// TwinCAT 3 PLC project PLC
// ProgramVersion: 3.1.4024.0
// libraries:
//   EfficientIO Communicator, * (EfficientIO)
//   EfficientIO ModbusTCP, * (EfficientIO)
//   Lynus Energy Basic, * (Lynus AG)
//   Lynus Persistent Data V1, * (Lynus AG)
//   Tc2_ModbusSrv, * (Beckhoff Automation GmbH)
//   Tc2_Standard, * (Beckhoff Automation GmbH)
//   Tc2_System, * (Beckhoff Automation GmbH)
//   Tc2_Utilities, * (Beckhoff Automation GmbH)
//   Tc3_Module, * (Beckhoff Automation GmbH)
//   Lynus Standards,1.0.0.1,Lynus AG
// project tree:
//   / FastTask.TcTTO, MiddleTask.TcTTO, SlowTask.TcTTO
//   FB/ FB_Symo_PV_Inverter_FLOAT_1_DM_1_Inverter_1.TcPOU
//   POUs/ prgComEffIO.TcPOU, prgEM.TcPOU, prgPersistent.TcPOU, prgPV.TcPOU, prgRWEffIO.TcPOU, prgVarEffIO.TcPOU
// real-time tasks:
//   TASK FastTask: cycle T#5ms, priority 19, ADS port 351
//   TASK SlowTask: cycle T#20ms, priority 21, ADS port 352
//   TASK MiddleTask: cycle T#10ms, priority 20, ADS port 353
// I/O:
//   DEVICE Gerät 2 (CX-BK)
//     Box 1 (CX-BK)
// variable links:
//   PLC/PLC Instance <-> Device 2 (CX-BK)/Box 1 (CX-BK)
//     MiddleTask Inputs/prgEM.fbEM1.fbKL3403.byStateCH1 <-> Term 2 (KL3403)/Channel 1/Status
//     MiddleTask Inputs/prgEM.fbEM1.fbKL3403.byStateCH2 <-> Term 2 (KL3403)/Channel 2/Status
//     MiddleTask Inputs/prgEM.fbEM1.fbKL3403.byStateCH3 <-> Term 2 (KL3403)/Channel 3/Status
//     MiddleTask Inputs/prgEM.fbEM2.fbKL3403.byStateCH1 <-> Term 3 (KL3403)/Channel 1/Status
//     MiddleTask Inputs/prgEM.fbEM2.fbKL3403.byStateCH2 <-> Term 3 (KL3403)/Channel 2/Status
//     MiddleTask Inputs/prgEM.fbEM2.fbKL3403.byStateCH3 <-> Term 3 (KL3403)/Channel 3/Status
//     MiddleTask Inputs/prgEM.fbEM3.fbKL3403.byStateCH1 <-> Term 4 (KL3403)/Channel 1/Status
//     MiddleTask Inputs/prgEM.fbEM3.fbKL3403.byStateCH2 <-> Term 4 (KL3403)/Channel 2/Status
//     MiddleTask Inputs/prgEM.fbEM3.fbKL3403.byStateCH3 <-> Term 4 (KL3403)/Channel 3/Status
//     MiddleTask Inputs/prgEM.fbEM4.fbKL3403.byStateCH1 <-> Term 5 (KL3403)/Channel 1/Status
//     MiddleTask Inputs/prgEM.fbEM4.fbKL3403.byStateCH2 <-> Term 5 (KL3403)/Channel 2/Status
//     MiddleTask Inputs/prgEM.fbEM4.fbKL3403.byStateCH3 <-> Term 5 (KL3403)/Channel 3/Status
//     MiddleTask Inputs/prgEM.fbEM5.fbKL3403.byStateCH1 <-> Term 6 (KL3403)/Channel 1/Status
//     MiddleTask Inputs/prgEM.fbEM5.fbKL3403.byStateCH2 <-> Term 6 (KL3403)/Channel 2/Status
//     MiddleTask Inputs/prgEM.fbEM5.fbKL3403.byStateCH3 <-> Term 6 (KL3403)/Channel 3/Status
//     MiddleTask Inputs/prgEM.fbEM6.fbKL3403.byStateCH1 <-> Term 7 (KL3403)/Channel 1/Status
//     MiddleTask Inputs/prgEM.fbEM6.fbKL3403.byStateCH2 <-> Term 7 (KL3403)/Channel 2/Status
//     MiddleTask Inputs/prgEM.fbEM6.fbKL3403.byStateCH3 <-> Term 7 (KL3403)/Channel 3/Status
//     MiddleTask Inputs/prgEM.fbEM7.fbKL3403.byStateCH1 <-> Term 8 (KL3403)/Channel 1/Status
//     MiddleTask Inputs/prgEM.fbEM7.fbKL3403.byStateCH2 <-> Term 8 (KL3403)/Channel 2/Status
//     MiddleTask Inputs/prgEM.fbEM7.fbKL3403.byStateCH3 <-> Term 8 (KL3403)/Channel 3/Status
//     MiddleTask Inputs/prgEM.fbEM8.fbKL3403.byStateCH1 <-> Term 9 (KL3403)/Channel 1/Status
//     MiddleTask Inputs/prgEM.fbEM8.fbKL3403.byStateCH2 <-> Term 9 (KL3403)/Channel 2/Status
//     MiddleTask Inputs/prgEM.fbEM8.fbKL3403.byStateCH3 <-> Term 9 (KL3403)/Channel 3/Status
//     MiddleTask Inputs/prgEM.fbEM9.fbKL3403.byStateCH1 <-> Term 10 (KL3403)/Channel 1/Status
//     MiddleTask Inputs/prgEM.fbEM9.fbKL3403.byStateCH2 <-> Term 10 (KL3403)/Channel 2/Status
//     MiddleTask Inputs/prgEM.fbEM9.fbKL3403.byStateCH3 <-> Term 10 (KL3403)/Channel 3/Status
//     MiddleTask Inputs/prgEM.fbEM1.fbKL3403.iDataInCH1 <-> Term 2 (KL3403)/Channel 1/Daten Ein
//     MiddleTask Inputs/prgEM.fbEM1.fbKL3403.iDataInCH2 <-> Term 2 (KL3403)/Channel 2/Daten Ein
//     MiddleTask Inputs/prgEM.fbEM1.fbKL3403.iDataInCH3 <-> Term 2 (KL3403)/Channel 3/Daten Ein
//     MiddleTask Inputs/prgEM.fbEM2.fbKL3403.iDataInCH1 <-> Term 3 (KL3403)/Channel 1/Daten Ein
//     MiddleTask Inputs/prgEM.fbEM2.fbKL3403.iDataInCH2 <-> Term 3 (KL3403)/Channel 2/Daten Ein
//     MiddleTask Inputs/prgEM.fbEM2.fbKL3403.iDataInCH3 <-> Term 3 (KL3403)/Channel 3/Daten Ein
//     MiddleTask Inputs/prgEM.fbEM3.fbKL3403.iDataInCH1 <-> Term 4 (KL3403)/Channel 1/Daten Ein
//     MiddleTask Inputs/prgEM.fbEM3.fbKL3403.iDataInCH2 <-> Term 4 (KL3403)/Channel 2/Daten Ein
//     MiddleTask Inputs/prgEM.fbEM3.fbKL3403.iDataInCH3 <-> Term 4 (KL3403)/Channel 3/Daten Ein
//     MiddleTask Inputs/prgEM.fbEM4.fbKL3403.iDataInCH1 <-> Term 5 (KL3403)/Channel 1/Daten Ein
//     MiddleTask Inputs/prgEM.fbEM4.fbKL3403.iDataInCH2 <-> Term 5 (KL3403)/Channel 2/Daten Ein
//     MiddleTask Inputs/prgEM.fbEM4.fbKL3403.iDataInCH3 <-> Term 5 (KL3403)/Channel 3/Daten Ein
//     MiddleTask Inputs/prgEM.fbEM5.fbKL3403.iDataInCH1 <-> Term 6 (KL3403)/Channel 1/Daten Ein
//     MiddleTask Inputs/prgEM.fbEM5.fbKL3403.iDataInCH2 <-> Term 6 (KL3403)/Channel 2/Daten Ein
//     MiddleTask Inputs/prgEM.fbEM5.fbKL3403.iDataInCH3 <-> Term 6 (KL3403)/Channel 3/Daten Ein
//     MiddleTask Inputs/prgEM.fbEM6.fbKL3403.iDataInCH1 <-> Term 7 (KL3403)/Channel 1/Daten Ein
//     MiddleTask Inputs/prgEM.fbEM6.fbKL3403.iDataInCH2 <-> Term 7 (KL3403)/Channel 2/Daten Ein
//     MiddleTask Inputs/prgEM.fbEM6.fbKL3403.iDataInCH3 <-> Term 7 (KL3403)/Channel 3/Daten Ein
//     MiddleTask Inputs/prgEM.fbEM7.fbKL3403.iDataInCH1 <-> Term 8 (KL3403)/Channel 1/Daten Ein
//     MiddleTask Inputs/prgEM.fbEM7.fbKL3403.iDataInCH2 <-> Term 8 (KL3403)/Channel 2/Daten Ein
//     MiddleTask Inputs/prgEM.fbEM7.fbKL3403.iDataInCH3 <-> Term 8 (KL3403)/Channel 3/Daten Ein
//     MiddleTask Inputs/prgEM.fbEM8.fbKL3403.iDataInCH1 <-> Term 9 (KL3403)/Channel 1/Daten Ein
//     MiddleTask Inputs/prgEM.fbEM8.fbKL3403.iDataInCH2 <-> Term 9 (KL3403)/Channel 2/Daten Ein
//     MiddleTask Inputs/prgEM.fbEM8.fbKL3403.iDataInCH3 <-> Term 9 (KL3403)/Channel 3/Daten Ein
//     MiddleTask Inputs/prgEM.fbEM9.fbKL3403.iDataInCH1 <-> Term 10 (KL3403)/Channel 1/Daten Ein
//     MiddleTask Inputs/prgEM.fbEM9.fbKL3403.iDataInCH2 <-> Term 10 (KL3403)/Channel 2/Daten Ein
//     MiddleTask Inputs/prgEM.fbEM9.fbKL3403.iDataInCH3 <-> Term 10 (KL3403)/Channel 3/Daten Ein
//     MiddleTask Inputs/prgEM.fbKBusState.uiKBusState_OUT <-> Inputs/State
//     MiddleTask Outputs/prgEM.fbEM1.fbKL3403.byCntrCH1 <-> Term 2 (KL3403)/Channel 1/Kontrolle
//     MiddleTask Outputs/prgEM.fbEM1.fbKL3403.byCntrCH2 <-> Term 2 (KL3403)/Channel 2/Kontrolle
//     MiddleTask Outputs/prgEM.fbEM1.fbKL3403.byCntrCH3 <-> Term 2 (KL3403)/Channel 3/Kontrolle
//     MiddleTask Outputs/prgEM.fbEM2.fbKL3403.byCntrCH1 <-> Term 3 (KL3403)/Channel 1/Kontrolle
//     MiddleTask Outputs/prgEM.fbEM2.fbKL3403.byCntrCH2 <-> Term 3 (KL3403)/Channel 2/Kontrolle
//     MiddleTask Outputs/prgEM.fbEM2.fbKL3403.byCntrCH3 <-> Term 3 (KL3403)/Channel 3/Kontrolle
//     MiddleTask Outputs/prgEM.fbEM3.fbKL3403.byCntrCH1 <-> Term 4 (KL3403)/Channel 1/Kontrolle
//     MiddleTask Outputs/prgEM.fbEM3.fbKL3403.byCntrCH2 <-> Term 4 (KL3403)/Channel 2/Kontrolle
//     MiddleTask Outputs/prgEM.fbEM3.fbKL3403.byCntrCH3 <-> Term 4 (KL3403)/Channel 3/Kontrolle
//     MiddleTask Outputs/prgEM.fbEM4.fbKL3403.byCntrCH1 <-> Term 5 (KL3403)/Channel 1/Kontrolle
//     MiddleTask Outputs/prgEM.fbEM4.fbKL3403.byCntrCH2 <-> Term 5 (KL3403)/Channel 2/Kontrolle
//     MiddleTask Outputs/prgEM.fbEM4.fbKL3403.byCntrCH3 <-> Term 5 (KL3403)/Channel 3/Kontrolle
//     MiddleTask Outputs/prgEM.fbEM5.fbKL3403.byCntrCH1 <-> Term 6 (KL3403)/Channel 1/Kontrolle
//     MiddleTask Outputs/prgEM.fbEM5.fbKL3403.byCntrCH2 <-> Term 6 (KL3403)/Channel 2/Kontrolle
//     MiddleTask Outputs/prgEM.fbEM5.fbKL3403.byCntrCH3 <-> Term 6 (KL3403)/Channel 3/Kontrolle
//     MiddleTask Outputs/prgEM.fbEM6.fbKL3403.byCntrCH1 <-> Term 7 (KL3403)/Channel 1/Kontrolle
//     MiddleTask Outputs/prgEM.fbEM6.fbKL3403.byCntrCH2 <-> Term 7 (KL3403)/Channel 2/Kontrolle
//     MiddleTask Outputs/prgEM.fbEM6.fbKL3403.byCntrCH3 <-> Term 7 (KL3403)/Channel 3/Kontrolle
//     MiddleTask Outputs/prgEM.fbEM7.fbKL3403.byCntrCH1 <-> Term 8 (KL3403)/Channel 1/Kontrolle
//     MiddleTask Outputs/prgEM.fbEM7.fbKL3403.byCntrCH2 <-> Term 8 (KL3403)/Channel 2/Kontrolle
//     MiddleTask Outputs/prgEM.fbEM7.fbKL3403.byCntrCH3 <-> Term 8 (KL3403)/Channel 3/Kontrolle
//     MiddleTask Outputs/prgEM.fbEM8.fbKL3403.byCntrCH1 <-> Term 9 (KL3403)/Channel 1/Kontrolle
//     MiddleTask Outputs/prgEM.fbEM8.fbKL3403.byCntrCH2 <-> Term 9 (KL3403)/Channel 2/Kontrolle
//     MiddleTask Outputs/prgEM.fbEM8.fbKL3403.byCntrCH3 <-> Term 9 (KL3403)/Channel 3/Kontrolle
//     MiddleTask Outputs/prgEM.fbEM9.fbKL3403.byCntrCH1 <-> Term 10 (KL3403)/Channel 1/Kontrolle
//     MiddleTask Outputs/prgEM.fbEM9.fbKL3403.byCntrCH2 <-> Term 10 (KL3403)/Channel 2/Kontrolle
//     MiddleTask Outputs/prgEM.fbEM9.fbKL3403.byCntrCH3 <-> Term 10 (KL3403)/Channel 3/Kontrolle

CONFIGURATION PLC
    RESOURCE PLC ON TwinCAT3
        TASK FastTask(INTERVAL := T#5ms, PRIORITY := 19);
        TASK MiddleTask(INTERVAL := T#10ms, PRIORITY := 20);
        TASK SlowTask(INTERVAL := T#20ms, PRIORITY := 21);
        PROGRAM prgVarEffIO WITH FastTask : prgVarEffIO;
        PROGRAM prgRWEffIO WITH FastTask : prgRWEffIO;
        PROGRAM prgPersistent WITH FastTask : prgPersistent;
        PROGRAM prgEM WITH MiddleTask : prgEM;
        PROGRAM prgPV WITH MiddleTask : prgPV;
        PROGRAM prgComEffIO WITH SlowTask : prgComEffIO;
    END_RESOURCE
END_CONFIGURATION

// ---- POUs/prgVarEffIO.TcPOU
PROGRAM prgVarEffIO
VAR
	fbVar		: FB_VarInfo;
END_VAR

fbVar(
	bReadInfo:= , 
	eTMCFile:= eSelectTMCFile.eDontUseTMCFile, 
	eSavePositionTMCFile:= eSavePositionOnPLC.ePostionHardDisk, 
	udiCounterFoundVariables=> , 
	bError=> , 
	bBusy=> , 
	byProgress=> , 
	udiErrorCodeOut=> , 
	eErrorVarInfo_Out=> , 
	sVarWithError=> );
fbVar();
fbVar();

END_PROGRAM

// ---- POUs/prgRWEffIO.TcPOU
PROGRAM prgRWEffIO
VAR
	fbRW1		: FB_ReadWrite_V2;
	fbRW2		: FB_ReadWrite;
	fbRW3		: FB_ReadWrite;
	fbRW4		: FB_ReadWrite;
	i: INT;
	x: INT:=1;
END_VAR

fbRW1(	eUploadType := eSelectDataUploadType.e_Change_Intervall5min,
		bBusy=> , 
		bError=> , 
		udiErrorCodeOut=> , 
		eErrorReadWrite_Out=> );

fbRW2();
fbRW3();
fbRW4();

(*
FOR i:= 1 TO x BY 1 DO
	fbRW1();
	
END_FOR
*)

END_PROGRAM

// ---- POUs/prgPersistent.TcPOU
PROGRAM prgPersistent
VAR
	fbUSV		: FB_WritePersistentData_CX81xx;
	fb_Reboot		: NT_reboot;
	m_Reboot		: BOOL:=FALSE;
	ton_Auto_Reboot_Delay: Ton;
END_VAR

fbUSV(
	eSaveModeData:= eUSVSaveMode.eSaveWhenPowerfail, 
	bLoadPersistentDataOk=> , 
	bPowerFailDetect=> , 
	bError=> , 
	bySaveProcess=> , 
	dwStorageLast24h=> , 
	udiErrorCode=> );
	
		
fb_Reboot(	netid := '',
			delay := 2,
			start := m_Reboot OR ton_Auto_Reboot_Delay.Q);
			
ton_Auto_Reboot_Delay( 	In:= NOT prgComEffIO.fbCom.bConnected,
						PT := T#10M);

END_PROGRAM

// ---- POUs/prgComEffIO.TcPOU
PROGRAM prgComEffIO
VAR
	fbCom		: FB_MqttCommunicator_V2;
END_VAR

fbCom(
	bConnect:= TRUE, 
	strAuthkey := 'EIO08031879806',
	sUserName:= '0c3f05a0-7dc5-40a2-afb3-e4500c155bc7', 			
	sUserPassword:= '792aca21-1d48-4069-8bd7-51e04ad34ff6', 		
	eSavePositionCertificate:= eSavePositionOnPLC.ePostionHardDisk, 
	bConnected=> , 
	bError=> , 
	hrErrorCode=> , 
	eConnectionState=> , 
	eErrorMessage_Out=> );

END_PROGRAM

// ---- POUs/prgEM.TcPOU
PROGRAM prgEM
VAR
	fbKBusState		: FB_K_Bus_State;
	fbEM1			: FB_EM_Beckhoff_KL3403;
	fbEM1Counter	: FB_EnergyCounter;
	fbEM2			: FB_EM_Beckhoff_KL3403;
	fbEM2Counter	: FB_EnergyCounter;
	fbEM3			: FB_EM_Beckhoff_KL3403;
	fbEM3Counter	: FB_EnergyCounter;
	fbEM4			: FB_EM_Beckhoff_KL3403;
	fbEM4Counter	: FB_EnergyCounter;
	fbEM5			: FB_EM_Beckhoff_KL3403;
	fbEM5Counter	: FB_EnergyCounter;
	fbEM6			: FB_EM_Beckhoff_KL3403;
	fbEM6Counter	: FB_EnergyCounter;
	fbEM7			: FB_EM_Beckhoff_KL3403;
	fbEM7Counter	: FB_EnergyCounter;
	fbEM8			: FB_EM_Beckhoff_KL3403;
	fbEM8Counter	: FB_EnergyCounter;
	fbEM9			: FB_EM_Beckhoff_KL3403;
	fbEM9Counter	: FB_EnergyCounter;
	
	lrPowerEM1		: LREAL;						//{#lynus.ag#()}
	lrPowerEM2		: LREAL;						//{#lynus.ag#()}
	lrPowerEM3		: LREAL;						//{#lynus.ag#()}
	lrPowerEM4		: LREAL;						//{#lynus.ag#()}
	lrPowerEM5		: LREAL;						//{#lynus.ag#()}
	lrPowerEM6		: LREAL;						//{#lynus.ag#()}
	lrPowerEM7		: LREAL;						//{#lynus.ag#()}
	lrPowerEM8		: LREAL;						//{#lynus.ag#()}
	lrPowerEM9		: LREAL;						//{#lynus.ag#()}
	lrPowerEM9_Production	: LREAL;						//{#lynus.ag#()}
	lrPowerEM9_Consumption	: LREAL;						//{#lynus.ag#()}
	lr_InputVoltage_L1N		: LREAL;						//{#lynus.ag#()}
	lr_InputVoltage_L2N		: LREAL;						//{#lynus.ag#()}
	lr_InputVoltage_L3N		: LREAL;						//{#lynus.ag#()}
	lr_InputVoltage_L1L2	: LREAL;						//{#lynus.ag#()}
	lr_InputVoltage_L2L3	: LREAL;						//{#lynus.ag#()}
	lr_InputVoltage_L3L1	: LREAL;						//{#lynus.ag#()}
	lr_FrequencyEM1			: LREAL;						//{#lynus.ag#()}
	lr_CurrentL1EM1			: LREAL;						//{#lynus.ag#()}
	lr_CurrentL2EM1			: LREAL;						//{#lynus.ag#()}
	lr_CurrentL3EM1			: LREAL;						//{#lynus.ag#()}
	lrPower_RestAltbau		: LREAL;						//{#lynus.ag#()}
	lrPower_RestNeubau		: LREAL;						//{#lynus.ag#()}
	lrPower_FirmaGesamt		: LREAL;						//{#lynus.ag#()}
	fbRest_Altbau_Counter	: FB_EnergyCounter;
	fbRest_Neubau_Counter	: FB_EnergyCounter;
	fbFirmaGesamt_Counter	: FB_EnergyCounter;

END_VAR
VAR_INPUT
	uiCurrentTransformerRatio_EM1	:UINT:=300;			
	uiCurrentTransformerRatio_EM2	:UINT:=250;			
	uiCurrentTransformerRatio_EM3	:UINT:=250;
	uiCurrentTransformerRatio_EM4	:UINT:=200;
	uiCurrentTransformerRatio_EM5	:UINT:=100;
	uiCurrentTransformerRatio_EM6	:UINT:=150;
	uiCurrentTransformerRatio_EM7	:UINT:=1250;
	uiCurrentTransformerRatio_EM8	:UINT:=500;
	uiCurrentTransformerRatio_EM9	:UINT:=1000;
	mtest: BOOL;

END_VAR
VAR PERSISTENT
	lrCounterEM1	: LREAL;						//{#lynus.ag#()}
	lrCounterEM2	: LREAL;						//{#lynus.ag#()}
	lrCounterEM3	: LREAL;						//{#lynus.ag#()}
	lrCounterEM4	: LREAL;						//{#lynus.ag#()}
	lrCounterEM5	: LREAL;						//{#lynus.ag#()}
	lrCounterEM6	: LREAL;						//{#lynus.ag#()}
	lrCounterEM7	: LREAL;						//{#lynus.ag#()}
	lrCounterEM8	: LREAL;						//{#lynus.ag#()}
	lrCounterEM9	: LREAL;						//{#lynus.ag#()}
	lrCounter_Grid_Prod	: LREAL;						//{#lynus.ag#()}
	lrCounter_Grid_Cons	: LREAL;						//{#lynus.ag#()}
	lrCounterRestAltbau	: LREAL;						//{#lynus.ag#()}
	lrCounterRestNeubau	: LREAL;						//{#lynus.ag#()}
	lrCounterFirmaGesamt: LREAL;						//{#lynus.ag#()}
END_VAR

fbKBusState(	uiKBusState_OUT=> , 
				b_Kbus_notOk=> , 
				word_ErrorCount=> );


fbEM1(
	bEnable:= TRUE, 
	bChannel1Invers:= FALSE,
	bChannel2Invers:= FALSE,
	bChannel3Invers:= FALSE,
	uiCurrentTransformerRatioL1:= uiCurrentTransformerRatio_EM1, 
	uiCurrentTransformerRatioL2:= uiCurrentTransformerRatio_EM1, 
	uiCurrentTransformerRatioL3:= uiCurrentTransformerRatio_EM1, 
	uiKBusState_IN:= fbKBusState.uiKBusState_OUT, 
	stDataEMPower=> , 
	stDataEMCounter=> , 
	stDataEMPowerRealTime=> , 
	stDataEMCounterRealTime=> , 
	diNrOfEM_OUT=> );

lrPowerEM1 := fbEM1.stDataEMPower.lrPowerTotal;	
lr_InputVoltage_L1N := fbEM1.stDataEMPower.lrVoltageL1N;
lr_InputVoltage_L2N := fbEM1.stDataEMPower.lrVoltageL2N;
lr_InputVoltage_L3N := fbEM1.stDataEMPower.lrVoltageL3N;
lr_InputVoltage_L1L2 := fbEM1.stDataEMPower.lrVoltageL1L2;
lr_InputVoltage_L2L3 := fbEM1.stDataEMPower.lrVoltageL2L3;
lr_InputVoltage_L3L1 := fbEM1.stDataEMPower.lrVoltageL3L1;
lr_FrequencyEM1		:= fbEM1.stDataEMPower.lrFrequency;
lr_CurrentL1EM1		:= fbEM1.stDataEMPower.lrCurrentL1;
lr_CurrentL2EM1		:= fbEM1.stDataEMPower.lrCurrentL2;
lr_CurrentL3EM1		:= fbEM1.stDataEMPower.lrCurrentL3;

fbEM1Counter(
	byActiveTariff:= 1, 
	lrPowerInput:= lrPowerEM1, 
	lrTotalCounterEnergy_Consumption=> , 
	lrTotalCounterEnergy_Production=> , 
	lrCounterEnergyT1_Consumption=> , 
	lrCounterEnergyT2_Consumption=> , 
	lrCounterEnergyT1_Production=> , 
	lrCounterEnergyT2_Production=> );
	
IF fbEM1Counter.lrTotalCounterEnergy_Consumption > lrCounterEM1 THEN  	
	lrCounterEM1 := fbEM1Counter.lrTotalCounterEnergy_Consumption;
END_IF


fbEM2(
	bEnable:= TRUE, 
	bChannel1Invers:= FALSE,
	bChannel2Invers:= FALSE,
	bChannel3Invers:= FALSE,
	uiCurrentTransformerRatioL1:= uiCurrentTransformerRatio_EM2, 
	uiCurrentTransformerRatioL2:= uiCurrentTransformerRatio_EM2, 
	uiCurrentTransformerRatioL3:= uiCurrentTransformerRatio_EM2, 
	uiKBusState_IN:= fbKBusState.uiKBusState_OUT, 
	stDataEMPower=> , 
	stDataEMCounter=> , 
	stDataEMPowerRealTime=> , 
	stDataEMCounterRealTime=> , 
	diNrOfEM_OUT=> );

lrPowerEM2 := fbEM2.stDataEMPower.lrPowerTotal;	

fbEM2Counter(
	byActiveTariff:= 1, 
	lrPowerInput:= lrPowerEM2, 
	lrTotalCounterEnergy_Consumption=> , 
	lrTotalCounterEnergy_Production=> , 
	lrCounterEnergyT1_Consumption=> , 
	lrCounterEnergyT2_Consumption=> , 
	lrCounterEnergyT1_Production=> , 
	lrCounterEnergyT2_Production=> );
	
IF fbEM2Counter.lrTotalCounterEnergy_Consumption > lrCounterEM2 THEN  	
	lrCounterEM2 := fbEM2Counter.lrTotalCounterEnergy_Consumption;
END_IF


fbEM3(
	bEnable:= TRUE, 
	bChannel1Invers:= FALSE,
	bChannel2Invers:= FALSE,
	bChannel3Invers:= FALSE,
	uiCurrentTransformerRatioL1:= uiCurrentTransformerRatio_EM3, 
	uiCurrentTransformerRatioL2:= uiCurrentTransformerRatio_EM3, 
	uiCurrentTransformerRatioL3:= uiCurrentTransformerRatio_EM3, 
	uiKBusState_IN:= fbKBusState.uiKBusState_OUT, 
	stDataEMPower=> , 
	stDataEMCounter=> , 
	stDataEMPowerRealTime=> , 
	stDataEMCounterRealTime=> , 
	diNrOfEM_OUT=> );

lrPowerEM3 := fbEM3.stDataEMPower.lrPowerTotal;	

fbEM3Counter(
	byActiveTariff:= 1, 
	lrPowerInput:= lrPowerEM3, 
	lrTotalCounterEnergy_Consumption=> , 
	lrTotalCounterEnergy_Production=> , 
	lrCounterEnergyT1_Consumption=> , 
	lrCounterEnergyT2_Consumption=> , 
	lrCounterEnergyT1_Production=> , 
	lrCounterEnergyT2_Production=> );
	
IF fbEM3Counter.lrTotalCounterEnergy_Consumption > lrCounterEM3 THEN  	
	lrCounterEM3 := fbEM3Counter.lrTotalCounterEnergy_Consumption;
END_IF

fbEM4(
	bEnable:= TRUE, 
	bChannel1Invers:= FALSE,
	bChannel2Invers:= FALSE,
	bChannel3Invers:= FALSE,
	uiCurrentTransformerRatioL1:= uiCurrentTransformerRatio_EM4, 
	uiCurrentTransformerRatioL2:= uiCurrentTransformerRatio_EM4, 
	uiCurrentTransformerRatioL3:= uiCurrentTransformerRatio_EM4, 
	uiKBusState_IN:= fbKBusState.uiKBusState_OUT, 
	stDataEMPower=> , 
	stDataEMCounter=> , 
	stDataEMPowerRealTime=> , 
	stDataEMCounterRealTime=> , 
	diNrOfEM_OUT=> );

lrPowerEM4 := fbEM4.stDataEMPower.lrPowerTotal;	

fbEM4Counter(
	byActiveTariff:= 1, 
	lrPowerInput:= lrPowerEM4, 
	lrTotalCounterEnergy_Consumption=> , 
	lrTotalCounterEnergy_Production=> , 
	lrCounterEnergyT1_Consumption=> , 
	lrCounterEnergyT2_Consumption=> , 
	lrCounterEnergyT1_Production=> , 
	lrCounterEnergyT2_Production=> );
	
IF fbEM4Counter.lrTotalCounterEnergy_Consumption > lrCounterEM4 THEN  	
	lrCounterEM4 := fbEM4Counter.lrTotalCounterEnergy_Consumption;
END_IF

fbEM5(
	bEnable:= TRUE, 
	bChannel1Invers:= FALSE,
	bChannel2Invers:= FALSE,
	bChannel3Invers:= FALSE,
	uiCurrentTransformerRatioL1:= uiCurrentTransformerRatio_EM5, 
	uiCurrentTransformerRatioL2:= uiCurrentTransformerRatio_EM5, 
	uiCurrentTransformerRatioL3:= uiCurrentTransformerRatio_EM5, 
	uiKBusState_IN:= fbKBusState.uiKBusState_OUT, 
	stDataEMPower=> , 
	stDataEMCounter=> , 
	stDataEMPowerRealTime=> , 
	stDataEMCounterRealTime=> , 
	diNrOfEM_OUT=> );

lrPowerEM5 := fbEM5.stDataEMPower.lrPowerTotal;	

fbEM5Counter(
	byActiveTariff:= 1, 
	lrPowerInput:= lrPowerEM5, 
	lrTotalCounterEnergy_Consumption=> , 
	lrTotalCounterEnergy_Production=> , 
	lrCounterEnergyT1_Consumption=> , 
	lrCounterEnergyT2_Consumption=> , 
	lrCounterEnergyT1_Production=> , 
	lrCounterEnergyT2_Production=> );
	
IF fbEM5Counter.lrTotalCounterEnergy_Consumption > lrCounterEM5 THEN  	
	lrCounterEM5 := fbEM5Counter.lrTotalCounterEnergy_Consumption;
END_IF

fbEM6(
	bEnable:= TRUE, 
	bChannel1Invers:= FALSE,
	bChannel2Invers:= FALSE,
	bChannel3Invers:= FALSE,
	uiCurrentTransformerRatioL1:= uiCurrentTransformerRatio_EM6, 
	uiCurrentTransformerRatioL2:= uiCurrentTransformerRatio_EM6, 
	uiCurrentTransformerRatioL3:= uiCurrentTransformerRatio_EM6, 
	uiKBusState_IN:= fbKBusState.uiKBusState_OUT, 
	stDataEMPower=> , 
	stDataEMCounter=> , 
	stDataEMPowerRealTime=> , 
	stDataEMCounterRealTime=> , 
	diNrOfEM_OUT=> );

lrPowerEM6 := fbEM6.stDataEMPower.lrPowerTotal;	

fbEM6Counter(
	byActiveTariff:= 1, 
	lrPowerInput:= lrPowerEM6, 
	lrTotalCounterEnergy_Consumption=> , 
	lrTotalCounterEnergy_Production=> , 
	lrCounterEnergyT1_Consumption=> , 
	lrCounterEnergyT2_Consumption=> , 
	lrCounterEnergyT1_Production=> , 
	lrCounterEnergyT2_Production=> );
	
IF fbEM6Counter.lrTotalCounterEnergy_Consumption > lrCounterEM6 THEN  	
	lrCounterEM6 := fbEM6Counter.lrTotalCounterEnergy_Consumption;
END_IF

fbEM7(
	bEnable:= TRUE, 
	bChannel1Invers:= FALSE,
	bChannel2Invers:= FALSE,
	bChannel3Invers:= FALSE,
	uiCurrentTransformerRatioL1:= uiCurrentTransformerRatio_EM7, 
	uiCurrentTransformerRatioL2:= uiCurrentTransformerRatio_EM7, 
	uiCurrentTransformerRatioL3:= uiCurrentTransformerRatio_EM7, 
	uiKBusState_IN:= fbKBusState.uiKBusState_OUT, 
	stDataEMPower=> , 
	stDataEMCounter=> , 
	stDataEMPowerRealTime=> , 
	stDataEMCounterRealTime=> , 
	diNrOfEM_OUT=> );

lrPowerEM7 := fbEM7.stDataEMPower.lrPowerTotal;	

fbEM7Counter(
	byActiveTariff:= 1, 
	lrPowerInput:= lrPowerEM7, 
	lrTotalCounterEnergy_Consumption=> , 
	lrTotalCounterEnergy_Production=> , 
	lrCounterEnergyT1_Consumption=> , 
	lrCounterEnergyT2_Consumption=> , 
	lrCounterEnergyT1_Production=> , 
	lrCounterEnergyT2_Production=> );
	
IF fbEM7Counter.lrTotalCounterEnergy_Consumption > lrCounterEM7 THEN  	
	lrCounterEM7 := fbEM7Counter.lrTotalCounterEnergy_Consumption;
END_IF

fbEM8(
	bEnable:= TRUE, 
	bChannel1Invers:= FALSE,
	bChannel2Invers:= FALSE,
	bChannel3Invers:= FALSE,
	uiCurrentTransformerRatioL1:= uiCurrentTransformerRatio_EM8, 
	uiCurrentTransformerRatioL2:= uiCurrentTransformerRatio_EM8, 
	uiCurrentTransformerRatioL3:= uiCurrentTransformerRatio_EM8, 
	uiKBusState_IN:= fbKBusState.uiKBusState_OUT, 
	stDataEMPower=> , 
	stDataEMCounter=> , 
	stDataEMPowerRealTime=> , 
	stDataEMCounterRealTime=> , 
	diNrOfEM_OUT=> );

lrPowerEM8 := fbEM8.stDataEMPower.lrPowerTotal;	

fbEM8Counter(
	byActiveTariff:= 1, 
	lrPowerInput:= lrPowerEM8, 
	lrTotalCounterEnergy_Consumption=> , 
	lrTotalCounterEnergy_Production=> , 
	lrCounterEnergyT1_Consumption=> , 
	lrCounterEnergyT2_Consumption=> , 
	lrCounterEnergyT1_Production=> , 
	lrCounterEnergyT2_Production=> );
	
IF fbEM8Counter.lrTotalCounterEnergy_Consumption > lrCounterEM8 THEN  	
	lrCounterEM8 := fbEM8Counter.lrTotalCounterEnergy_Consumption;
END_IF

fbEM9(
	bEnable:= TRUE, 
	bChannel1Invers:= FALSE,
	bChannel2Invers:= FALSE,
	bChannel3Invers:= FALSE,
	uiCurrentTransformerRatioL1:= uiCurrentTransformerRatio_EM9, 
	uiCurrentTransformerRatioL2:= uiCurrentTransformerRatio_EM9, 
	uiCurrentTransformerRatioL3:= uiCurrentTransformerRatio_EM9, 
	uiKBusState_IN:= fbKBusState.uiKBusState_OUT, 
	stDataEMPower=> , 
	stDataEMCounter=> , 
	stDataEMPowerRealTime=> , 
	stDataEMCounterRealTime=> , 
	diNrOfEM_OUT=> );

lrPowerEM9 := fbEM9.stDataEMPower.lrPowerTotal;	

IF lrPowerEM9<= 0 THEN
	lrPowerEM9_Production :=  lrPowerEM9;
	lrPowerEM9_Consumption := 0;
ELSE
	lrPowerEM9_Production :=  0;
	lrPowerEM9_Consumption := lrPowerEM9;
END_IF

fbEM9Counter(
	byActiveTariff:= 1, 
	lrPowerInput:= lrPowerEM9, 
	lrTotalCounterEnergy_Consumption=> , 
	lrTotalCounterEnergy_Production=> , 
	lrCounterEnergyT1_Consumption=> , 
	lrCounterEnergyT2_Consumption=> , 
	lrCounterEnergyT1_Production=> , 
	lrCounterEnergyT2_Production=> );
	
IF fbEM9Counter.lrTotalCounterEnergy_Consumption > lrCounterEM9 THEN  	
	lrCounterEM9 := fbEM9Counter.lrTotalCounterEnergy_Consumption;
	lrCounter_Grid_Cons	:= fbEM9Counter.lrTotalCounterEnergy_Consumption;
END_IF

IF fbEM9Counter.lrTotalCounterEnergy_Production > lrCounter_Grid_Prod THEN  	
	lrCounter_Grid_Prod := fbEM9Counter.lrTotalCounterEnergy_Production;
END_IF

lrPower_RestAltbau := lrPowerEM8 - lrPowerEM1 - lrPowerEM2 - lrPowerEM3 - lrPowerEM4 + prgPV.lrPowerPV;
lrPower_RestAltbau := LIMIT(0,lrPower_RestAltbau,lrPower_RestAltbau);
lrPower_RestNeubau := lrPowerEM9 - lrPowerEM8 - lrPowerEM5 - lrPowerEM6;
lrPower_RestNeubau := LIMIT(0,lrPower_RestNeubau,lrPower_RestNeubau);

lrPower_FirmaGesamt := lrPowerEM9 + prgPV.lrPowerPV;


fbRest_Altbau_Counter(
	byActiveTariff:= 1, 
	lrPowerInput:= lrPower_RestAltbau, 
	lrTotalCounterEnergy_Consumption=> , 
	lrTotalCounterEnergy_Production=> , 
	lrCounterEnergyT1_Consumption=> , 
	lrCounterEnergyT2_Consumption=> , 
	lrCounterEnergyT1_Production=> , 
	lrCounterEnergyT2_Production=> );
	
IF fbRest_Altbau_Counter.lrTotalCounterEnergy_Consumption > lrCounterRestAltbau THEN  	
	lrCounterRestAltbau := fbRest_Altbau_Counter.lrTotalCounterEnergy_Consumption;
END_IF


fbRest_Neubau_Counter(
	byActiveTariff:= 1, 
	lrPowerInput:= lrPower_RestNeubau, 
	lrTotalCounterEnergy_Consumption=> , 
	lrTotalCounterEnergy_Production=> , 
	lrCounterEnergyT1_Consumption=> , 
	lrCounterEnergyT2_Consumption=> , 
	lrCounterEnergyT1_Production=> , 
	lrCounterEnergyT2_Production=> );
	
IF fbRest_Neubau_Counter.lrTotalCounterEnergy_Consumption > lrCounterRestNeubau THEN  	
	lrCounterRestNeubau := fbRest_Neubau_Counter.lrTotalCounterEnergy_Consumption;
END_IF


fbFirmaGesamt_Counter(
	byActiveTariff:= 1, 
	lrPowerInput:= lrPower_FirmaGesamt, 
	lrTotalCounterEnergy_Consumption=> , 
	lrTotalCounterEnergy_Production=> , 
	lrCounterEnergyT1_Consumption=> , 
	lrCounterEnergyT2_Consumption=> , 
	lrCounterEnergyT1_Production=> , 
	lrCounterEnergyT2_Production=> );
	
IF fbFirmaGesamt_Counter.lrTotalCounterEnergy_Consumption > lrCounterFirmaGesamt THEN  	
	lrCounterFirmaGesamt := fbFirmaGesamt_Counter.lrTotalCounterEnergy_Consumption;
END_IF

END_PROGRAM

// ---- POUs/prgPV.TcPOU
PROGRAM prgPV
VAR
	fbPV_1					: FB_Symo_PV_Inverter_float_1_DM_1_Inverter_1;
	fbPV_2					: FB_Symo_PV_Inverter_float_1_DM_1_Inverter_1;
	fbPV_3					: FB_Symo_PV_Inverter_float_1_DM_1_Inverter_1;
	fbPV_4					: FB_Symo_PV_Inverter_float_1_DM_1_Inverter_1;
	fbPV_5					: FB_Symo_PV_Inverter_float_1_DM_1_Inverter_1;
	fbPV_6					: FB_Symo_PV_Inverter_float_1_DM_1_Inverter_1;
	fbPV_7					: FB_Symo_PV_Inverter_float_1_DM_1_Inverter_1;
	fbPV_8					: FB_Symo_PV_Inverter_float_1_DM_1_Inverter_1;
	lrPowerPV				: LREAL;				//{#lynus.ag#()}
	lrPowerPV_1				: LREAL;				//{#lynus.ag#()}
	lrPowerPV_2				: LREAL;				//{#lynus.ag#()}
	lrPowerPV_3				: LREAL;				//{#lynus.ag#()}
	lrPowerPV_4				: LREAL;				//{#lynus.ag#()}
	lrPowerPV_5				: LREAL;				//{#lynus.ag#()}
	lrPowerPV_6				: LREAL;				//{#lynus.ag#()}
	lrPowerPV_7				: LREAL;				//{#lynus.ag#()}
	lrPowerPV_8				: LREAL;				//{#lynus.ag#()}
	fbCounterPV_1			: FB_EnergyCounter;
	fbCounterPV_2			: FB_EnergyCounter;
	fbCounterPV_3			: FB_EnergyCounter;
	fbCounterPV_4			: FB_EnergyCounter;
	fbCounterPV_5			: FB_EnergyCounter;
	fbCounterPV_6			: FB_EnergyCounter;
	fbCounterPV_7			: FB_EnergyCounter;
	fbCounterPV_8			: FB_EnergyCounter;
	fbCounterPV				: FB_EnergyCounter;
END_VAR
VAR PERSISTENT
	lrCounterPV_1	: LREAL;						//{#lynus.ag#()}
	lrCounterPV_2	: LREAL;						//{#lynus.ag#()}
	lrCounterPV_3	: LREAL;						//{#lynus.ag#()}
	lrCounterPV_4	: LREAL;						//{#lynus.ag#()}
	lrCounterPV_5	: LREAL;						//{#lynus.ag#()}
	lrCounterPV_6	: LREAL;						//{#lynus.ag#()}
	lrCounterPV_7	: LREAL;						//{#lynus.ag#()}
	lrCounterPV_8	: LREAL;						//{#lynus.ag#()}
	lrCounterPV		: LREAL;						//{#lynus.ag#()}
	m_Enable_PV1: BOOL:= TRUE;
	m_Enable_PV2: BOOL:= true;
	m_Enable_PV3: BOOL:= true;
	m_Enable_PV4: BOOL:= true;
	m_Enable_PV5: BOOL:= true;
	m_Enable_PV6: BOOL:= true;
	m_Enable_PV7: BOOL:= true;
	m_Enable_PV8: BOOL:= true;	

END_VAR

fbPV_1(
	bEnable:= TRUE, 
	sIPAdress:= '192.168.10.12', 
	byUnitID_Inverter:=3 , 
	stDataSymo10=> , 
	stDataEMPower_PV=> , 
	stDataEMCounter_PV=> , 
	diNrOfEM_OUT_PV=> );
lrPowerPV_1 := fbPV_1.stDataEMPower_PV.lrPowerTotal;
fbPV_2(
	bEnable:= m_Enable_PV2, 
	sIPAdress:= '192.168.10.13', 
	byUnitID_Inverter:=2 , 
	stDataSymo10=> , 
	stDataEMPower_PV=> , 
	stDataEMCounter_PV=> , 
	diNrOfEM_OUT_PV=> );
lrPowerPV_2 := fbPV_2.stDataEMPower_PV.lrPowerTotal;
fbPV_3(
	bEnable:= m_Enable_PV3, 
	sIPAdress:= '192.168.10.14', 
	byUnitID_Inverter:=5 , 
	stDataSymo10=> , 
	stDataEMPower_PV=> , 
	stDataEMCounter_PV=> , 
	diNrOfEM_OUT_PV=> );
lrPowerPV_3 := fbPV_3.stDataEMPower_PV.lrPowerTotal;
fbPV_4(
	bEnable:= m_Enable_PV4, 
	sIPAdress:= '192.168.10.15', 
	byUnitID_Inverter:=4 , 
	stDataSymo10=> , 
	stDataEMPower_PV=> , 
	stDataEMCounter_PV=> , 
	diNrOfEM_OUT_PV=> );
lrPowerPV_4 := fbPV_4.stDataEMPower_PV.lrPowerTotal;
fbPV_5(
	bEnable:= m_Enable_PV5, 
	sIPAdress:= '192.168.10.16', 
	byUnitID_Inverter:=1 , 
	stDataSymo10=> , 
	stDataEMPower_PV=> , 
	stDataEMCounter_PV=> , 
	diNrOfEM_OUT_PV=> );
lrPowerPV_5 := fbPV_5.stDataEMPower_PV.lrPowerTotal;
fbPV_6(
	bEnable:= m_Enable_PV6, 
	sIPAdress:= '192.168.10.17', 
	byUnitID_Inverter:=1 , 
	stDataSymo10=> , 
	stDataEMPower_PV=> , 
	stDataEMCounter_PV=> , 
	diNrOfEM_OUT_PV=> );
lrPowerPV_6 := fbPV_6.stDataEMPower_PV.lrPowerTotal;
fbPV_7(
	bEnable:= m_Enable_PV7, 
	sIPAdress:= '192.168.10.18', 
	byUnitID_Inverter:=1 , 
	stDataSymo10=> , 
	stDataEMPower_PV=> , 
	stDataEMCounter_PV=> , 
	diNrOfEM_OUT_PV=> );
lrPowerPV_7 := fbPV_7.stDataEMPower_PV.lrPowerTotal;
fbPV_8(
	bEnable:= m_Enable_PV8, 
	sIPAdress:= '192.168.10.19', 
	byUnitID_Inverter:=1 , 
	stDataSymo10=> , 
	stDataEMPower_PV=> , 
	stDataEMCounter_PV=> , 
	diNrOfEM_OUT_PV=> );
lrPowerPV_8 := fbPV_8.stDataEMPower_PV.lrPowerTotal;

lrPowerPV := lrPowerPV_1 + lrPowerPV_2 + lrPowerPV_3 + lrPowerPV_4 + lrPowerPV_5 + lrPowerPV_6 + lrPowerPV_7 + lrPowerPV_8;


// kWh Counters

fbCounterPV_1(
	byActiveTariff:= 1, 
	lrPowerInput:= lrPowerPV_1, 
	lrTotalCounterEnergy_Consumption=> , 
	lrTotalCounterEnergy_Production=> , 
	lrCounterEnergyT1_Consumption=> , 
	lrCounterEnergyT2_Consumption=> , 
	lrCounterEnergyT1_Production=> , 
	lrCounterEnergyT2_Production=> );
	
IF fbCounterPV_1.lrTotalCounterEnergy_Consumption > lrCounterPV_1 THEN  	
	lrCounterPV_1 := fbCounterPV_1.lrTotalCounterEnergy_Consumption;
END_IF

fbCounterPV_2(
	byActiveTariff:= 1, 
	lrPowerInput:= lrPowerPV_2, 
	lrTotalCounterEnergy_Consumption=> , 
	lrTotalCounterEnergy_Production=> , 
	lrCounterEnergyT1_Consumption=> , 
	lrCounterEnergyT2_Consumption=> , 
	lrCounterEnergyT1_Production=> , 
	lrCounterEnergyT2_Production=> );
	
IF fbCounterPV_2.lrTotalCounterEnergy_Consumption > lrCounterPV_2 THEN  	
	lrCounterPV_2 := fbCounterPV_2.lrTotalCounterEnergy_Consumption;
END_IF

fbCounterPV_3(
	byActiveTariff:= 1, 
	lrPowerInput:= lrPowerPV_3, 
	lrTotalCounterEnergy_Consumption=> , 
	lrTotalCounterEnergy_Production=> , 
	lrCounterEnergyT1_Consumption=> , 
	lrCounterEnergyT2_Consumption=> , 
	lrCounterEnergyT1_Production=> , 
	lrCounterEnergyT2_Production=> );
	
IF fbCounterPV_3.lrTotalCounterEnergy_Consumption > lrCounterPV_3 THEN  	
	lrCounterPV_3 := fbCounterPV_3.lrTotalCounterEnergy_Consumption;
END_IF

fbCounterPV_4(
	byActiveTariff:= 1, 
	lrPowerInput:= lrPowerPV_4, 
	lrTotalCounterEnergy_Consumption=> , 
	lrTotalCounterEnergy_Production=> , 
	lrCounterEnergyT1_Consumption=> , 
	lrCounterEnergyT2_Consumption=> , 
	lrCounterEnergyT1_Production=> , 
	lrCounterEnergyT2_Production=> );
	
IF fbCounterPV_4.lrTotalCounterEnergy_Consumption > lrCounterPV_4 THEN  	
	lrCounterPV_4 := fbCounterPV_4.lrTotalCounterEnergy_Consumption;
END_IF

fbCounterPV_5(
	byActiveTariff:= 1, 
	lrPowerInput:= lrPowerPV_5, 
	lrTotalCounterEnergy_Consumption=> , 
	lrTotalCounterEnergy_Production=> , 
	lrCounterEnergyT1_Consumption=> , 
	lrCounterEnergyT2_Consumption=> , 
	lrCounterEnergyT1_Production=> , 
	lrCounterEnergyT2_Production=> );
	
IF fbCounterPV_5.lrTotalCounterEnergy_Consumption > lrCounterPV_5 THEN  	
	lrCounterPV_5 := fbCounterPV_5.lrTotalCounterEnergy_Consumption;
END_IF

fbCounterPV_6(
	byActiveTariff:= 1, 
	lrPowerInput:= lrPowerPV_6, 
	lrTotalCounterEnergy_Consumption=> , 
	lrTotalCounterEnergy_Production=> , 
	lrCounterEnergyT1_Consumption=> , 
	lrCounterEnergyT2_Consumption=> , 
	lrCounterEnergyT1_Production=> , 
	lrCounterEnergyT2_Production=> );
	
IF fbCounterPV_6.lrTotalCounterEnergy_Consumption > lrCounterPV_6 THEN  	
	lrCounterPV_6 := fbCounterPV_6.lrTotalCounterEnergy_Consumption;
END_IF

fbCounterPV_7(
	byActiveTariff:= 1, 
	lrPowerInput:= lrPowerPV_7, 
	lrTotalCounterEnergy_Consumption=> , 
	lrTotalCounterEnergy_Production=> , 
	lrCounterEnergyT1_Consumption=> , 
	lrCounterEnergyT2_Consumption=> , 
	lrCounterEnergyT1_Production=> , 
	lrCounterEnergyT2_Production=> );
	
IF fbCounterPV_7.lrTotalCounterEnergy_Consumption > lrCounterPV_7 THEN  	
	lrCounterPV_7 := fbCounterPV_7.lrTotalCounterEnergy_Consumption;
END_IF

fbCounterPV_8(
	byActiveTariff:= 1, 
	lrPowerInput:= lrPowerPV_8, 
	lrTotalCounterEnergy_Consumption=> , 
	lrTotalCounterEnergy_Production=> , 
	lrCounterEnergyT1_Consumption=> , 
	lrCounterEnergyT2_Consumption=> , 
	lrCounterEnergyT1_Production=> , 
	lrCounterEnergyT2_Production=> );
	
IF fbCounterPV_8.lrTotalCounterEnergy_Consumption > lrCounterPV_8 THEN  	
	lrCounterPV_8 := fbCounterPV_8.lrTotalCounterEnergy_Consumption;
END_IF

fbCounterPV(
	byActiveTariff:= 1, 
	lrPowerInput:= lrPowerPV, 
	lrTotalCounterEnergy_Consumption=> , 
	lrTotalCounterEnergy_Production=> , 
	lrCounterEnergyT1_Consumption=> , 
	lrCounterEnergyT2_Consumption=> , 
	lrCounterEnergyT1_Production=> , 
	lrCounterEnergyT2_Production=> );
	
IF fbCounterPV.lrTotalCounterEnergy_Consumption > lrCounterPV THEN  	
	lrCounterPV := fbCounterPV.lrTotalCounterEnergy_Consumption;
END_IF

END_PROGRAM

// ---- FB/FB_Symo_PV_Inverter_FLOAT_1_DM_1_Inverter_1.TcPOU
{attribute 'hide_all_locals'}
FUNCTION_BLOCK FB_Symo_PV_Inverter_FLOAT_1_DM_1_Inverter_1
VAR_INPUT PERSISTENT
	bEnable						: BOOL;												//True = Function is enabled, FALSE = Function is dissabled, no new Data
	sIPAdress					: STRING(15);										//IP Adress from the Inverter
	byUnitID_Inverter			: BYTE;												//Unit ID fromt the Inverter (1 to 247)
END_VAR
VAR_OUTPUT
	stDataSymo10				: ST_Symo_PV_OutData;								//Output structure with Data from Symo 10
	stDataEMPower_PV			: ST_ElectricMeter_Output_Power;					//Output structure with Data from Electric Meter PV (Power Data)
	stDataEMCounter_PV			: ST_ElectricMeter_Output_Counter;					//Output structure with Data from Electric Meter PV (Counter Data)
	diNrOfEM_OUT_PV				: DINT;												//Active Number from the Electric Meter for using on other functions
END_VAR
VAR
	fbElMeter					: FB_ElectricMeter;									//Electric Meter Function 
	fbNumberDevice				: FB_NumberOfDevice;								//Function block to calcualte the number of the Device
	fbConvertEnergyRegister		: FB_CV_WORD_TO_DWORD;								//Convert function
	fbMBRead_FC3				: FB_MBReadRegs;									//Modbus Read Function (FC3)
	timDelay					: TON;												//Timer for Delay between Requests
	timTimeout					: TON;												//Timer for Timeout
	timDissableFunctions		: TON;												//Timer to dissable the Function after Lynus_Standards.Constants_General.tTimeDissableLynusFunctions Days without connection to the Lynus Cloud
	timResetConnectionOnGVL		: TON;												//Timer to try reset the connection Flag on the GVL. (When somebody delete the Connection Function and make only a onlinechange)
	FPEnable					: R_TRIG;											//Internal positive Edge
	FPError_FC_3				: R_TRIG;											//Internal positive Edge
	PD_String					: FB_PersistentData_String;							//Function to save persistent data 
	stFloat						: ST_UN_FLOAT_CONVERT_DWORD_REAL;					//Convert the Float Raw Value
	arrBuffer_FC3				: ARRAY[1..47] OF WORD;								//Buffer with Data from FC3
	arrPD						: ARRAY[1..2] OF FB_PersistentData_Number;			//Function to save persistent data 
	byWaitInStep				: BYTE;												//Wait in Step before start to clean data on PLC
	iStateGVLData				: INT;												//State machine to handle the data on the GVL
	iStateModbus				: INT;												//State variable for Statemachine
	iStateModbus_CP				: INT;												//Compare State variable
	diCounterForGVL				: DINT;												//Counter to clean old data on GVL
	lrCheckValue				: LREAL;											//Internal Value to check the value before convert
END_VAR

//Creator : Kai Ebensperger
//Company : Lynus AG
//Date : 28.04.2021
//Version : 1.0.0.0

//With this function its possible to read out values from the Symo 10 PV Inverter from the factory Fronius
//This Function read out the Values from 1 Fronius Datamanager with maximal 1 Inverter.
//The protocol to the Inverter is Modbus TCP
//Versions that are supported : 1.1.5-0
//Attention. To access the registers, an offset of 1 must always be subtracted. Register 40001 would then be on register 40000.
//This Function use the FLOAT Format

//NOTE for diNr.....Designation => 
//_IN = Here Data come in from other Functions or go out to other functions about the GVL
//_OUT = Here Data go out to other functions about the GVL

(*------------------------------------------------------------------------------------------General Input Part---------------------------------------------------------------------------------------------*)

//Check limitation
byUnitID_Inverter := LIMIT(1,byUnitID_Inverter,247);

(*-------------------------------------------------------------Calcualte the number of EM System---------------------------------------------------------------*)

fbNumberDevice(
	diActualNumberOfDevices:= Lynus_Standards.GVL_Energy.stNumberOfDevices.diNumberOfElectricMeters, 
	diMaxNumberOfDevices:= Constants_Energy.diMaxNumberOfElectricMeters, 
	udiCounterOnlineChange:= TwinCAT_SystemInfoVarList._AppInfo.OnlineChangeCnt, 
	bNumberIsCalculatet=> , 
	bFPNumberIsCalculatet=> , 
	bOnlineChange=> , 
	diNumberForThisDevice=> diNrOfEM_OUT_PV, 
	diNumberOfTotalDevices=> );

//Write new Numer on GVL
IF fbNumberDevice.bFPNumberIsCalculatet THEN
	Lynus_Standards.GVL_Energy.stNumberOfDevices.diNumberOfElectricMeters := fbNumberDevice.diNumberOfTotalDevices;	
END_IF 

//Delete old Number on GVL
IF fbNumberDevice.bOnlineChange THEN 
	Lynus_Standards.GVL_Energy.stNumberOfDevices.diNumberOfElectricMeters := diNrOfEM_OUT_PV;	
		iStateGVLData := 1; 
END_IF

(*-------------------------------------------------------------Service from Backend is ready and check the connection to backen for dissabel/enable Function---------------------------------------------------------------*)

//Try to reset the variable for connection on the GVL. When all is normal then the Lynus Mqtt connection function set this variable to true in the next cycle
//When we have no connection to the backend then after Lynus_Standards.Constants_General.tTimeDissableLynusFunctions days the Function is dissabled with all of his functionalities
timResetConnectionOnGVL(IN:= NOT timResetConnectionOnGVL.Q, PT:= T#1H, Q=> , ET=> );
	IF timResetConnectionOnGVL.Q THEN Lynus_Standards.GVL_Communicator.bStateConnectionToEnableFunctions := FALSE; END_IF
		IF NOT Lynus_Standards.GVL_Communicator.bStateConnectionToEnableFunctions THEN timDissableFunctions.IN := TRUE; ELSE timDissableFunctions.IN := FALSE; END_IF  
			timDissableFunctions(IN:= , PT:= Lynus_Standards.Constants_General.tTimeDissableLynusFunctions, Q=> , ET=> );
	
(*------------------------------------------------------------------------------------------State Machine---------------------------------------------------------------------------------------------*)
	
//Enable
FPEnable(CLK:= bEnable, Q=> );
	IF FPEnable.Q AND iStateModbus = 0 THEN iStateModbus := 1; END_IF
		IF NOT bEnable OR timDissableFunctions.Q THEN iStateModbus := 0; END_IF

//Timer for delay
timDelay(IN:= , PT:= T#100MS, Q=> , ET=> );	

//Timer for Timeout in Statemachine
	IF iStateModbus = iStateModbus_CP THEN timTimeout.IN := TRUE; ELSE timTimeout.IN := FALSE; END_IF
		IF iStateModbus = 0 THEN timTimeout.IN := FALSE; END_IF
timTimeout(IN:= , PT:= T#20S, Q=> , ET=> );	

//Statemachine
CASE iStateModbus OF
	
	0://Init Step
		iStateModbus_CP := iStateModbus;
			timDelay.IN := FALSE;
		
		stDataSymo10.bFunctionIsActive := FALSE;
			stDataSymo10.eOperatingStateInverter := E_Symo_PV_OperatingState.eNoDataReceived;
				fbMBRead_FC3.bExecute := FALSE;
					lrCheckValue := 0;
									
	1://Read out first Registers from 40072 to 40118
		stDataSymo10.bFunctionIsActive := TRUE;
			iStateModbus_CP := iStateModbus;
		
		fbMBRead_FC3.nQuantity := 47;
			fbMBRead_FC3.nMBAddr := 40071;
				fbMBRead_FC3.bExecute := TRUE;
					fbMBRead_FC3.nUnitID := byUnitID_Inverter;
			
		IF fbMBRead_FC3.bBusy THEN timDelay.IN := TRUE; END_IF
		
		//Wait for Delay, copy Data and then next step
		IF NOT fbMBRead_FC3.bBusy AND NOT fbMBRead_FC3.bError AND timDelay.Q THEN
			//Copy Data Current L1
			fbConvertEnergyRegister(wInputValue_1:= arrBuffer_FC3[3], wInputValue_2:= arrBuffer_FC3[4], eByteOrderForConvert:= eByteOrder.eBigEndian, dwOutputValue=> );
				stFloat.dwRawValue := fbConvertEnergyRegister.dwOutputValue;
					lrCheckValue := stFloat.rValueFloat;	
						IF lrCheckValue >= - 3.402823E+38 AND lrCheckValue <= 3.402823E+38 THEN 
							fbElMeter.lrCurrentL1 := lrCheckValue;
						ELSE
							iStateModbus := 300;
								stDataSymo10.eErrorState := E_Symo_PV_Error.eSymo10TooBigValueReceived;		
						END_IF
			//Copy Data Current L2
			fbConvertEnergyRegister(wInputValue_1:= arrBuffer_FC3[5], wInputValue_2:= arrBuffer_FC3[6], eByteOrderForConvert:= eByteOrder.eBigEndian, dwOutputValue=> );
				stFloat.dwRawValue := fbConvertEnergyRegister.dwOutputValue;
					lrCheckValue := stFloat.rValueFloat;	
						IF lrCheckValue >= - 3.402823E+38 AND lrCheckValue <= 3.402823E+38 THEN 
							fbElMeter.lrCurrentL2 := lrCheckValue;
						ELSE
							iStateModbus := 300;
								stDataSymo10.eErrorState := E_Symo_PV_Error.eSymo10TooBigValueReceived;		
						END_IF
			//Copy Data Current L3
			fbConvertEnergyRegister(wInputValue_1:= arrBuffer_FC3[7], wInputValue_2:= arrBuffer_FC3[8], eByteOrderForConvert:= eByteOrder.eBigEndian, dwOutputValue=> );
				stFloat.dwRawValue := fbConvertEnergyRegister.dwOutputValue;
					lrCheckValue := stFloat.rValueFloat;	
						IF lrCheckValue >= - 3.402823E+38 AND lrCheckValue <= 3.402823E+38 THEN 
							fbElMeter.lrCurrentL3 := lrCheckValue;
						ELSE
							iStateModbus := 300;
								stDataSymo10.eErrorState := E_Symo_PV_Error.eSymo10TooBigValueReceived;		
						END_IF
			//Copy Data Voltage L1-L2
			fbConvertEnergyRegister(wInputValue_1:= arrBuffer_FC3[9], wInputValue_2:= arrBuffer_FC3[10], eByteOrderForConvert:= eByteOrder.eBigEndian, dwOutputValue=> );
				stFloat.dwRawValue := fbConvertEnergyRegister.dwOutputValue;
					lrCheckValue := stFloat.rValueFloat;	
						IF lrCheckValue >= - 3.402823E+38 AND lrCheckValue <= 3.402823E+38 THEN 
							fbElMeter.lrVoltageL1L2 := lrCheckValue;
						ELSE
							iStateModbus := 300;
								stDataSymo10.eErrorState := E_Symo_PV_Error.eSymo10TooBigValueReceived;		
						END_IF
			//Copy Data Voltage L2-L3
			fbConvertEnergyRegister(wInputValue_1:= arrBuffer_FC3[11], wInputValue_2:= arrBuffer_FC3[12], eByteOrderForConvert:= eByteOrder.eBigEndian, dwOutputValue=> );
				stFloat.dwRawValue := fbConvertEnergyRegister.dwOutputValue;
					lrCheckValue := stFloat.rValueFloat;	
						IF lrCheckValue >= - 3.402823E+38 AND lrCheckValue <= 3.402823E+38 THEN 
							fbElMeter.lrVoltageL2L3 := lrCheckValue;
						ELSE
							iStateModbus := 300;
								stDataSymo10.eErrorState := E_Symo_PV_Error.eSymo10TooBigValueReceived;		
						END_IF
			//Copy Data Voltage L3-L1
			fbConvertEnergyRegister(wInputValue_1:= arrBuffer_FC3[13], wInputValue_2:= arrBuffer_FC3[14], eByteOrderForConvert:= eByteOrder.eBigEndian, dwOutputValue=> );
				stFloat.dwRawValue := fbConvertEnergyRegister.dwOutputValue;
					lrCheckValue := stFloat.rValueFloat;	
						IF lrCheckValue >= - 3.402823E+38 AND lrCheckValue <= 3.402823E+38 THEN 
							fbElMeter.lrVoltageL3L1 := lrCheckValue;
						ELSE
							iStateModbus := 300;
								stDataSymo10.eErrorState := E_Symo_PV_Error.eSymo10TooBigValueReceived;		
						END_IF
			//Copy Data Voltage L1-N
			fbConvertEnergyRegister(wInputValue_1:= arrBuffer_FC3[15], wInputValue_2:= arrBuffer_FC3[16], eByteOrderForConvert:= eByteOrder.eBigEndian, dwOutputValue=> );
				stFloat.dwRawValue := fbConvertEnergyRegister.dwOutputValue;
					lrCheckValue := stFloat.rValueFloat;	
						IF lrCheckValue >= - 3.402823E+38 AND lrCheckValue <= 3.402823E+38 THEN 
							fbElMeter.lrVoltageL1N := lrCheckValue;
						ELSE
							iStateModbus := 300;
								stDataSymo10.eErrorState := E_Symo_PV_Error.eSymo10TooBigValueReceived;		
						END_IF
			//Copy Data Voltage L2-N
			fbConvertEnergyRegister(wInputValue_1:= arrBuffer_FC3[17], wInputValue_2:= arrBuffer_FC3[18], eByteOrderForConvert:= eByteOrder.eBigEndian, dwOutputValue=> );
				stFloat.dwRawValue := fbConvertEnergyRegister.dwOutputValue;
					lrCheckValue := stFloat.rValueFloat;	
						IF lrCheckValue >= - 3.402823E+38 AND lrCheckValue <= 3.402823E+38 THEN 
							fbElMeter.lrVoltageL2N := lrCheckValue;
						ELSE
							iStateModbus := 300;
								stDataSymo10.eErrorState := E_Symo_PV_Error.eSymo10TooBigValueReceived;		
						END_IF
			//Copy Data Voltage L3-N
			fbConvertEnergyRegister(wInputValue_1:= arrBuffer_FC3[19], wInputValue_2:= arrBuffer_FC3[20], eByteOrderForConvert:= eByteOrder.eBigEndian, dwOutputValue=> );
				stFloat.dwRawValue := fbConvertEnergyRegister.dwOutputValue;
					lrCheckValue := stFloat.rValueFloat;	
						IF lrCheckValue >= - 3.402823E+38 AND lrCheckValue <= 3.402823E+38 THEN 
							fbElMeter.lrVoltageL3N := lrCheckValue;
						ELSE
							iStateModbus := 300;
								stDataSymo10.eErrorState := E_Symo_PV_Error.eSymo10TooBigValueReceived;		
						END_IF
			//Copy Data AC Power
			fbConvertEnergyRegister(wInputValue_1:= arrBuffer_FC3[21], wInputValue_2:= arrBuffer_FC3[22], eByteOrderForConvert:= eByteOrder.eBigEndian, dwOutputValue=> );
				stFloat.dwRawValue := fbConvertEnergyRegister.dwOutputValue;
					lrCheckValue := stFloat.rValueFloat;	
						IF lrCheckValue >= - 3.402823E+38 AND lrCheckValue <= 3.402823E+38 THEN 
							fbElMeter.lrPowerTotal := lrCheckValue;
						ELSE
							iStateModbus := 300;
								stDataSymo10.eErrorState := E_Symo_PV_Error.eSymo10TooBigValueReceived;		
						END_IF
			//Copy Data Frequency
			fbConvertEnergyRegister(wInputValue_1:= arrBuffer_FC3[23], wInputValue_2:= arrBuffer_FC3[24], eByteOrderForConvert:= eByteOrder.eBigEndian, dwOutputValue=> );
				stFloat.dwRawValue := fbConvertEnergyRegister.dwOutputValue;
					lrCheckValue := stFloat.rValueFloat;	
						IF lrCheckValue >= - 3.402823E+38 AND lrCheckValue <= 3.402823E+38 THEN 
							fbElMeter.lrFrequency := lrCheckValue;
						ELSE
							iStateModbus := 300;
								stDataSymo10.eErrorState := E_Symo_PV_Error.eSymo10TooBigValueReceived;		
						END_IF
			//Copy Data Apparent Power
			fbConvertEnergyRegister(wInputValue_1:= arrBuffer_FC3[25], wInputValue_2:= arrBuffer_FC3[26], eByteOrderForConvert:= eByteOrder.eBigEndian, dwOutputValue=> );
				stFloat.dwRawValue := fbConvertEnergyRegister.dwOutputValue;
					lrCheckValue := stFloat.rValueFloat;	
						IF lrCheckValue >= - 3.402823E+38 AND lrCheckValue <= 3.402823E+38 THEN 
							fbElMeter.lrApparentPowerTotal := lrCheckValue;
						ELSE
							iStateModbus := 300;
								stDataSymo10.eErrorState := E_Symo_PV_Error.eSymo10TooBigValueReceived;		
						END_IF
			//Copy Data Reactive Power
			fbConvertEnergyRegister(wInputValue_1:= arrBuffer_FC3[27], wInputValue_2:= arrBuffer_FC3[28], eByteOrderForConvert:= eByteOrder.eBigEndian, dwOutputValue=> );
				stFloat.dwRawValue := fbConvertEnergyRegister.dwOutputValue;
					lrCheckValue := stFloat.rValueFloat;	
						IF lrCheckValue >= - 3.402823E+38 AND lrCheckValue <= 3.402823E+38 THEN 
							fbElMeter.lrReactivePowerTotal := lrCheckValue;
						ELSE
							iStateModbus := 300;
								stDataSymo10.eErrorState := E_Symo_PV_Error.eSymo10TooBigValueReceived;		
						END_IF
			//Copy Data AC production Energy
			fbConvertEnergyRegister(wInputValue_1:= arrBuffer_FC3[31], wInputValue_2:= arrBuffer_FC3[32], eByteOrderForConvert:= eByteOrder.eBigEndian, dwOutputValue=> );
				stFloat.dwRawValue := fbConvertEnergyRegister.dwOutputValue;
					lrCheckValue := stFloat.rValueFloat;	
						IF lrCheckValue >= - 3.402823E+38 AND lrCheckValue <= 3.402823E+38 THEN 
							fbElMeter.lrCounterEnergyT1_Production := lrCheckValue / 1000;
								fbElMeter.lrTotalCounterEnergy_Production := fbElMeter.lrCounterEnergyT1_Production;
						ELSE
							iStateModbus := 300;
								stDataSymo10.eErrorState := E_Symo_PV_Error.eSymo10TooBigValueReceived;		
						END_IF
			//Operating State		
			IF arrBuffer_FC3[47] = 1 THEN stDataSymo10.eOperatingStateInverter := E_Symo_PV_OperatingState.eOff;
				ELSIF arrBuffer_FC3[47] = 2 THEN stDataSymo10.eOperatingStateInverter := E_Symo_PV_OperatingState.eSleeping;
				ELSIF arrBuffer_FC3[47] = 3 THEN stDataSymo10.eOperatingStateInverter := E_Symo_PV_OperatingState.eStartingUp;
				ELSIF arrBuffer_FC3[47] = 4 THEN stDataSymo10.eOperatingStateInverter := E_Symo_PV_OperatingState.eTrackingPowerPoint;
				ELSIF arrBuffer_FC3[47] = 5 THEN stDataSymo10.eOperatingStateInverter := E_Symo_PV_OperatingState.eForcedPowerReduction;
				ELSIF arrBuffer_FC3[47] = 6 THEN stDataSymo10.eOperatingStateInverter := E_Symo_PV_OperatingState.eShuttingDown;
				ELSIF arrBuffer_FC3[47] = 7 THEN stDataSymo10.eOperatingStateInverter := E_Symo_PV_OperatingState.eFaults;
				ELSIF arrBuffer_FC3[47] = 8 THEN stDataSymo10.eOperatingStateInverter := E_Symo_PV_OperatingState.eStandby;
				ELSE stDataSymo10.eOperatingStateInverter := E_Symo_PV_OperatingState.eNoDataReceived;
			END_IF
			//Next Step
			IF iStateModbus = 1 THEN
				fbMBRead_FC3.bExecute := FALSE;
					timDelay.IN := FALSE;
						iStateModbus := 2;
							stDataSymo10.bError := FALSE; 
								stDataSymo10.eErrorState := E_Symo_PV_Error.eNoError;
			END_IF
		END_IF
			
		//Error from Inverter
		IF NOT fbMBRead_FC3.bBusy AND NOT fbMBRead_FC3.bError AND timDelay.Q AND stDataSymo10.eOperatingStateInverter = E_Symo_PV_OperatingState.eFaults THEN
			iStateModbus := 300;
				stDataSymo10.eErrorState := E_Symo_PV_Error.eSymo10Error;
		END_IF
	 
		//Error or Timeout
		IF FPError_FC_3.Q OR timTimeout.Q THEN
			iStateModbus := 300;
				stDataSymo10.eErrorState := E_Symo_PV_Error.eModbusTCPError;
		END_IF

	2://Wait and back to 1 step
		iStateModbus_CP := iStateModbus;
		
			iStateModbus := 1;
				
	300://Error
		iStateModbus_CP := iStateModbus;
			timDelay.IN := FALSE;
				fbMBRead_FC3.bExecute := FALSE;
					stDataSymo10.bError := TRUE;
						iStateModbus := 1;				
							
END_CASE

(*------------------------------------------------------------------------------------------Modbus TCP Function---------------------------------------------------------------------------------------------*)

fbMBRead_FC3(sIPAddr:= sIPAdress, nTCPPort:= 502, cbLength:= SIZEOF(arrBuffer_FC3), pDestAddr:= ADR(arrBuffer_FC3), tTimeout:= T#10S );
	FPError_FC_3(CLK:= fbMBRead_FC3.bError, Q=> );

(*----------------------------------------------------------------------------------------Electric Meter Data----------------------------------------------------------------------------------------------*)

//Error and Warning
IF timDissableFunctions.Q THEN fbElMeter.bWarning := TRUE; fbElMeter.iWarningCode := 0; ELSE fbElMeter.bWarning := FALSE; END_IF   
	IF stDataSymo10.bError OR Lynus_Standards.GVL_Energy.stNumberOfDevices.diNumberOfElectricMeters > Constants_Energy.diMaxNumberOfElectricMeters THEN fbElMeter.bError := TRUE; ELSE fbElMeter.bError := FALSE; END_IF  

IF Lynus_Standards.GVL_Energy.stNumberOfDevices.diNumberOfElectricMeters > Constants_Energy.diMaxNumberOfElectricMeters THEN fbElMeter.iErrorCode := 1;
ELSIF stDataSymo10.bError THEN fbElMeter.iErrorCode := 0;
END_IF  

//Read Out Data done for EM Function
IF iStateModbus <> 2 THEN fbElMeter.bReadOutDataDone := TRUE; ELSE fbElMeter.bReadOutDataDone := FALSE; END_IF

//Function block for meter data
fbElMeter(
	bEnable:= bEnable AND NOT timDissableFunctions.Q, 
	bError:= , 
	bEnableReadOutFunction:= FALSE, 
	bWriteWithDelay:= TRUE,
	bPowerDataInvers:= TRUE, 
	bReadOutDataDone:= ,
	iTimeReadOutInterval:= , 
	iErrorCode:= , 
	iWarningCode:= , 
	lrTotalCounterEnergy_Consumption:= 0, 
	lrTotalCounterEnergy_Production:= , 
	lrCounterEnergyT1_Consumption:= 0, 
	lrCounterEnergyT2_Consumption:= 0, 
	lrCounterEnergyT1_Production:= , 
	lrCounterEnergyT2_Production:= 0, 
	lrCurrentL1:= , 
	lrVoltageL1N:= , 
	lrVoltageL1L2:= , 
	lrPowerL1:= 0, 
	lrCurrentL2:= , 
	lrVoltageL2N:= , 
	lrVoltageL2L3:= , 
	lrPowerL2:= 0, 
	lrCurrentL3:= , 
	lrVoltageL3N:= , 
	lrVoltageL3L1:= , 
	lrPowerL3:= 0, 
	lrPowerTotal:= , 
	lrFrequency:= , 
	lrReactivePowerTotal:= , 
	lrApparentPowerTotal:= , 
	tTimDelayOutput:= T#5S, 
	stDataEMOutPower=> , 
	stDataEMOutPowerDelay=> stDataEMPower_PV, 
	stDataEMOutCounter=> ,
	stDataEMOutCounterDelay=> stDataEMCounter_PV, 
	bReadOutMeter=> );

(*-----------------------------------------------------------Handle data to Global structure for the Electric Meter system-----------------------------------------------------------------*)

CASE iStateGVLData OF
	
	0://Init Step
		byWaitInStep := 0;
			diCounterForGVL := 1;
	
	1://Wait for 4 Steps before clean al Data on GVL
		byWaitInStep := byWaitInStep + 1;
			IF byWaitInStep >= 4 AND fbNumberDevice.bNumberIsCalculatet THEN iStateGVLData := 2; END_IF
				//To much Devices, back to the Init step
				IF byWaitInStep >= 4 AND NOT fbNumberDevice.bNumberIsCalculatet THEN iStateGVLData := 0; END_IF	
			
	2://Clear all Data in GVL
		Lynus_Standards.GVL_Energy.stDataElectricMeters[diCounterForGVL].bEnabled := FALSE;	
			Lynus_Standards.GVL_Energy.stDataElectricMeters[diCounterForGVL].byErrorWarning := 0;
				Lynus_Standards.GVL_Energy.stDataElectricMeters[diCounterForGVL].lrCounterEnergyT1_Consumption := 0;
					Lynus_Standards.GVL_Energy.stDataElectricMeters[diCounterForGVL].lrCounterEnergyT1_Production := 0;
						Lynus_Standards.GVL_Energy.stDataElectricMeters[diCounterForGVL].lrCounterEnergyT2_Consumption := 0;
							Lynus_Standards.GVL_Energy.stDataElectricMeters[diCounterForGVL].lrCounterEnergyT2_Production := 0;
								Lynus_Standards.GVL_Energy.stDataElectricMeters[diCounterForGVL].lrPower := 0;
									Lynus_Standards.GVL_Energy.stDataElectricMeters[diCounterForGVL].lrPowerConsumption := 0;
										Lynus_Standards.GVL_Energy.stDataElectricMeters[diCounterForGVL].lrPowerConsumption := 0;
											Lynus_Standards.GVL_Energy.stDataElectricMeters[diCounterForGVL].lrPowerProduction := 0;
												Lynus_Standards.GVL_Energy.stDataElectricMeters[diCounterForGVL].lrTotalCounterEnergy_Consumption := 0;
													Lynus_Standards.GVL_Energy.stDataElectricMeters[diCounterForGVL].lrTotalCounterEnergy_Production := 0;
		
		diCounterForGVL := diCounterForGVL + 1;
			diCounterForGVL := LIMIT(0,diCounterForGVL,Constants_Energy.diMaxNumberOfElectricMeters);
				//Back to the init step
				IF diCounterForGVL >= Constants_Energy.diMaxNumberOfElectricMeters THEN iStateGVLData := 0; END_IF

END_CASE 	 

IF diNrOfEM_OUT_PV > 0 AND fbNumberDevice.bNumberIsCalculatet THEN
	Lynus_Standards.GVL_Energy.stDataElectricMeters[diNrOfEM_OUT_PV].bEnabled := fbElMeter.stDataEMOutPower.bEnabled;
		Lynus_Standards.GVL_Energy.stDataElectricMeters[diNrOfEM_OUT_PV].byErrorWarning := fbElMeter.stDataEMOutPower.byErrorWarning;
			Lynus_Standards.GVL_Energy.stDataElectricMeters[diNrOfEM_OUT_PV].lrCounterEnergyT1_Consumption := fbElMeter.stDataEMOutCounter.lrCounterEnergyT1_Consumption;
				Lynus_Standards.GVL_Energy.stDataElectricMeters[diNrOfEM_OUT_PV].lrCounterEnergyT1_Production := fbElMeter.stDataEMOutCounter.lrCounterEnergyT1_Production;
					Lynus_Standards.GVL_Energy.stDataElectricMeters[diNrOfEM_OUT_PV].lrCounterEnergyT2_Consumption := fbElMeter.stDataEMOutCounter.lrCounterEnergyT2_Consumption;
						Lynus_Standards.GVL_Energy.stDataElectricMeters[diNrOfEM_OUT_PV].lrCounterEnergyT2_Production := fbElMeter.stDataEMOutCounter.lrCounterEnergyT2_Production;		
							Lynus_Standards.GVL_Energy.stDataElectricMeters[diNrOfEM_OUT_PV].lrPower := fbElMeter.stDataEMOutPower.lrPowerTotal;
								Lynus_Standards.GVL_Energy.stDataElectricMeters[diNrOfEM_OUT_PV].lrPowerConsumption := fbElMeter.stDataEMOutPower.lrPowerConsumption;
									Lynus_Standards.GVL_Energy.stDataElectricMeters[diNrOfEM_OUT_PV].lrPowerProduction := fbElMeter.stDataEMOutPower.lrPowerProduction;
										Lynus_Standards.GVL_Energy.stDataElectricMeters[diNrOfEM_OUT_PV].lrTotalCounterEnergy_Consumption := fbElMeter.stDataEMOutCounter.lrTotalCounterEnergy_Consumption;
											Lynus_Standards.GVL_Energy.stDataElectricMeters[diNrOfEM_OUT_PV].lrTotalCounterEnergy_Production := fbElMeter.stDataEMOutCounter.lrTotalCounterEnergy_Production;
END_IF

(*----------------------------------------------------------Save persistent data----------------------------------------------------------------*)

arrPD[1](lrValue:= BOOL_TO_LREAL(bEnable), bEventBasedActive=> );
arrPD[2](lrValue:= BYTE_TO_LREAL(byUnitID_Inverter), bEventBasedActive=> );
PD_String(sText:= sIPAdress, bEventBasedActive=> );

END_FUNCTION_BLOCK
